prgEM.stEL3443_IO.MDP5001_341_Input.MDP5001_341_L1_Status_Voltage_Sign_Bit 		:= MDP5001_341_L1_Status_Voltage_Sign_Bit;
prgEM.stEL3443_IO.MDP5001_341_Input.MDP5001_341_L1_Status_Overvoltage			:= MDP5001_341_L1_Status_Overvoltage;
prgEM.stEL3443_IO.MDP5001_341_Input.MDP5001_341_L1_Status_Overcurrent			:= MDP5001_341_L1_Status_Overcurrent;
prgEM.stEL3443_IO.MDP5001_341_Input.MDP5001_341_L1_Status_Inaccurate_Voltage	:= MDP5001_341_L1_Status_Inaccurate_Voltage;
prgEM.stEL3443_IO.MDP5001_341_Input.MDP5001_341_L1_Status_Inaccurate_Current	:= MDP5001_341_L1_Status_Inaccurate_Current;
prgEM.stEL3443_IO.MDP5001_341_Input.MDP5001_341_L1_Status_Voltage_Guard_Warning	:= MDP5001_341_L1_Status_Voltage_Guard_Warning;
prgEM.stEL3443_IO.MDP5001_341_Input.MDP5001_341_L1_Status_Voltage_Guard_Error	:= MDP5001_341_L1_Status_Voltage_Guard_Error;
prgEM.stEL3443_IO.MDP5001_341_Input.MDP5001_341_L1_Status_Current_Guard_Warning	:= MDP5001_341_L1_Status_Current_Guard_Warning;
prgEM.stEL3443_IO.MDP5001_341_Input.MDP5001_341_L1_Status_Current_Guard_Error	:= MDP5001_341_L1_Status_Current_Guard_Error;
prgEM.stEL3443_IO.MDP5001_341_Input.MDP5001_341_L1_Status_TxPDO_Toggle			:= MDP5001_341_L1_Status_TxPDO_Toggle;
prgEM.stEL3443_IO.MDP5001_341_Input.MDP5001_341_L1_Basic_Voltage				:= MDP5001_341_L1_Basic_Voltage;
prgEM.stEL3443_IO.MDP5001_341_Input.MDP5001_341_L1_Basic_Current				:= MDP5001_341_L1_Basic_Current;
prgEM.stEL3443_IO.MDP5001_341_Input.MDP5001_341_L1_Power_Active_Power			:= MDP5001_341_L1_Power_Active_Power;
prgEM.stEL3443_IO.MDP5001_341_Input.MDP5001_341_L1_Power_Apparent_Power			:= MDP5001_341_L1_Power_Apparent_Power;
prgEM.stEL3443_IO.MDP5001_341_Input.MDP5001_341_L1_Power_Reactive_Power			:= MDP5001_341_L1_Power_Reactive_Power;
prgEM.stEL3443_IO.MDP5001_341_Input.MDP5001_341_L1_Power_Power_Factor			:= MDP5001_341_L1_Power_Power_Factor;
prgEM.stEL3443_IO.MDP5001_341_Input.MDP5001_341_L2_Status_Voltage_Sign_Bit 		:= MDP5001_341_L2_Status_Voltage_Sign_Bit;
prgEM.stEL3443_IO.MDP5001_341_Input.MDP5001_341_L2_Status_Overvoltage			:= MDP5001_341_L2_Status_Overvoltage;
prgEM.stEL3443_IO.MDP5001_341_Input.MDP5001_341_L2_Status_Overcurrent			:= MDP5001_341_L2_Status_Overcurrent;
prgEM.stEL3443_IO.MDP5001_341_Input.MDP5001_341_L2_Status_Inaccurate_Voltage	:= MDP5001_341_L2_Status_Inaccurate_Voltage;
prgEM.stEL3443_IO.MDP5001_341_Input.MDP5001_341_L2_Status_Inaccurate_Current	:= MDP5001_341_L2_Status_Inaccurate_Current;
prgEM.stEL3443_IO.MDP5001_341_Input.MDP5001_341_L2_Status_Voltage_Guard_Warning	:= MDP5001_341_L2_Status_Voltage_Guard_Warning;
prgEM.stEL3443_IO.MDP5001_341_Input.MDP5001_341_L2_Status_Voltage_Guard_Error	:= MDP5001_341_L2_Status_Voltage_Guard_Error;
prgEM.stEL3443_IO.MDP5001_341_Input.MDP5001_341_L2_Status_Current_Guard_Warning	:= MDP5001_341_L2_Status_Current_Guard_Warning;
prgEM.stEL3443_IO.MDP5001_341_Input.MDP5001_341_L2_Status_Current_Guard_Error	:= MDP5001_341_L2_Status_Current_Guard_Error;
prgEM.stEL3443_IO.MDP5001_341_Input.MDP5001_341_L2_Status_TxPDO_Toggle			:= MDP5001_341_L2_Status_TxPDO_Toggle;
prgEM.stEL3443_IO.MDP5001_341_Input.MDP5001_341_L2_Basic_Voltage				:= MDP5001_341_L2_Basic_Voltage;
prgEM.stEL3443_IO.MDP5001_341_Input.MDP5001_341_L2_Basic_Current				:= MDP5001_341_L2_Basic_Current;
prgEM.stEL3443_IO.MDP5001_341_Input.MDP5001_341_L2_Power_Active_Power			:= MDP5001_341_L2_Power_Active_Power;
prgEM.stEL3443_IO.MDP5001_341_Input.MDP5001_341_L2_Power_Apparent_Power			:= MDP5001_341_L2_Power_Apparent_Power;
prgEM.stEL3443_IO.MDP5001_341_Input.MDP5001_341_L2_Power_Reactive_Power			:= MDP5001_341_L2_Power_Reactive_Power;
prgEM.stEL3443_IO.MDP5001_341_Input.MDP5001_341_L2_Power_Power_Factor			:= MDP5001_341_L2_Power_Power_Factor;
prgEM.stEL3443_IO.MDP5001_341_Input.MDP5001_341_L3_Status_Voltage_Sign_Bit 		:= MDP5001_341_L3_Status_Voltage_Sign_Bit;
prgEM.stEL3443_IO.MDP5001_341_Input.MDP5001_341_L3_Status_Overvoltage			:= MDP5001_341_L3_Status_Overvoltage;
prgEM.stEL3443_IO.MDP5001_341_Input.MDP5001_341_L3_Status_Overcurrent			:= MDP5001_341_L3_Status_Overcurrent;
prgEM.stEL3443_IO.MDP5001_341_Input.MDP5001_341_L3_Status_Inaccurate_Voltage	:= MDP5001_341_L3_Status_Inaccurate_Voltage;
prgEM.stEL3443_IO.MDP5001_341_Input.MDP5001_341_L3_Status_Inaccurate_Current	:= MDP5001_341_L3_Status_Inaccurate_Current;
prgEM.stEL3443_IO.MDP5001_341_Input.MDP5001_341_L3_Status_Voltage_Guard_Warning	:= MDP5001_341_L3_Status_Voltage_Guard_Warning;
prgEM.stEL3443_IO.MDP5001_341_Input.MDP5001_341_L3_Status_Voltage_Guard_Error	:= MDP5001_341_L3_Status_Voltage_Guard_Error;
prgEM.stEL3443_IO.MDP5001_341_Input.MDP5001_341_L3_Status_Current_Guard_Warning	:= MDP5001_341_L3_Status_Current_Guard_Warning;
prgEM.stEL3443_IO.MDP5001_341_Input.MDP5001_341_L3_Status_Current_Guard_Error	:= MDP5001_341_L3_Status_Current_Guard_Error;
prgEM.stEL3443_IO.MDP5001_341_Input.MDP5001_341_L3_Status_TxPDO_Toggle			:= MDP5001_341_L3_Status_TxPDO_Toggle;
prgEM.stEL3443_IO.MDP5001_341_Input.MDP5001_341_L3_Basic_Voltage				:= MDP5001_341_L3_Basic_Voltage;
prgEM.stEL3443_IO.MDP5001_341_Input.MDP5001_341_L3_Basic_Current				:= MDP5001_341_L3_Basic_Current;
prgEM.stEL3443_IO.MDP5001_341_Input.MDP5001_341_L3_Power_Active_Power			:= MDP5001_341_L3_Power_Active_Power;
prgEM.stEL3443_IO.MDP5001_341_Input.MDP5001_341_L3_Power_Apparent_Power			:= MDP5001_341_L3_Power_Apparent_Power;
prgEM.stEL3443_IO.MDP5001_341_Input.MDP5001_341_L3_Power_Reactive_Power			:= MDP5001_341_L3_Power_Reactive_Power;
prgEM.stEL3443_IO.MDP5001_341_Input.MDP5001_341_L3_Power_Power_Factor			:= MDP5001_341_L3_Power_Power_Factor;
prgEM.stEL3443_IO.MDP5001_341_Input.MDP5001_341_Total_Status_System_State		:= MDP5001_341_Total_Status_System_State  ;	
prgEM.stEL3443_IO.MDP5001_341_Input.MDP5001_341_Total_Status_Grid_Direction		:= MDP5001_341_Total_Status_Grid_Direction ;
prgEM.stEL3443_IO.MDP5001_341_Input.MDP5001_341_Total_Status_Frequency_Guard_Warning 		:= MDP5001_341_Total_Status_Frequency_Guard_Warning ;
prgEM.stEL3443_IO.MDP5001_341_Input.MDP5001_341_Total_Status_Frequency_Guard_Error 			:= MDP5001_341_Total_Status_Frequency_Guard_Error  ;
prgEM.stEL3443_IO.MDP5001_341_Input.MDP5001_341_Total_Status_Neutral_Current_Guard_Warning	:= MDP5001_341_Total_Status_Neutral_Current_Guard_Warning ;
prgEM.stEL3443_IO.MDP5001_341_Input.MDP5001_341_Total_Status_Neutral_Current_Guard_Error	:= MDP5001_341_Total_Status_Neutral_Current_Guard_Error;
prgEM.stEL3443_IO.MDP5001_341_Input.MDP5001_341_Total_Status_Active_Power_Guard_Warning		:= MDP5001_341_Total_Status_Active_Power_Guard_Warning ;
prgEM.stEL3443_IO.MDP5001_341_Input.MDP5001_341_Total_Status_Active_Power_Guard_Error		:= MDP5001_341_Total_Status_Active_Power_Guard_Error ;
prgEM.stEL3443_IO.MDP5001_341_Input.MDP5001_341_Total_Status_Apparent_Power_Guard_Warning	:= MDP5001_341_Total_Status_Apparent_Power_Guard_Warning ;
prgEM.stEL3443_IO.MDP5001_341_Input.MDP5001_341_Total_Status_Apparent_Power_Guard_Error		:= MDP5001_341_Total_Status_Apparent_Power_Guard_Error ;
prgEM.stEL3443_IO.MDP5001_341_Input.MDP5001_341_Total_Status_Power_Quality_Guard_Warning	:= MDP5001_341_Total_Status_Power_Quality_Guard_Warning ;
prgEM.stEL3443_IO.MDP5001_341_Input.MDP5001_341_Total_Status_Power_Quality_Guard_Error		:= MDP5001_341_Total_Status_Power_Quality_Guard_Error ;
prgEM.stEL3443_IO.MDP5001_341_Input.MDP5001_341_Total_Status_TxPDO_State					:= MDP5001_341_Total_Status_TxPDO_State ;
prgEM.stEL3443_IO.MDP5001_341_Input.MDP5001_341_Total_Status_TxPDO_Toggle					:= MDP5001_341_Total_Status_TxPDO_Toggle ;
prgEM.stEL3443_IO.MDP5001_341_Input.MDP5001_341_Total_Status_Power_Quality_Factor			:= MDP5001_341_Total_Status_Power_Quality_Factor ;
prgEM.stEL3443_IO.MDP5001_341_Input.MDP5001_341_Total_Basic_Frequency						:= MDP5001_341_Total_Basic_Frequency;
prgEM.stEL3443_IO.MDP5001_341_Input.MDP5001_341_Total_Basic_Power_Factor					:= MDP5001_341_Total_Basic_Power_Factor  ;
prgEM.stEL3443_IO.MDP5001_341_Input.MDP5001_341_Total_Basic_Calculated_Neutral_Line_Current	:= MDP5001_341_Total_Basic_Calculated_Neutral_Line_Current ;
prgEM.stEL3443_IO.MDP5001_341_Input.MDP5001_341_Total_Variant_Value_In_TxPDO_Toggle			:= MDP5001_341_Total_Variant_Value_In_TxPDO_Toggle ;
prgEM.stEL3443_IO.MDP5001_341_Input.MDP5001_341_Total_Variant_Value_In_Index_1_REAL			:= MDP5001_341_Total_Variant_Value_In_Index_1_REAL ;
prgEM.stEL3443_IO.MDP5001_341_Input.MDP5001_341_Total_Variant_Value_In_Value_1_REAL			:= MDP5001_341_Total_Variant_Value_In_Value_1_REAL ;
prgEM.stEL3443_IO.MDP5001_341_Input.MDP5001_341_Total_Variant_Value_In_Index_2_REAL			:= MDP5001_341_Total_Variant_Value_In_Index_2_REAL ;
prgEM.stEL3443_IO.MDP5001_341_Input.MDP5001_341_Total_Variant_Value_In_Value_2_REAL			:= MDP5001_341_Total_Variant_Value_In_Value_2_REAL ;
prgEM.stEL3443_IO.MDP5001_341_Input.MDP5001_341_Total_Variant_Value_In_Index_3_REAL			:= MDP5001_341_Total_Variant_Value_In_Index_3_REAL ;
prgEM.stEL3443_IO.MDP5001_341_Input.MDP5001_341_Total_Variant_Value_In_Value_3_REAL			:= MDP5001_341_Total_Variant_Value_In_Value_3_REAL ;
prgEM.stEL3443_IO.MDP5001_341_Input.MDP5001_341_Total_Variant_Value_In_Index_4_ULINT		:= MDP5001_341_Total_Variant_Value_In_Index_4_ULINT ;
prgEM.stEL3443_IO.MDP5001_341_Input.MDP5001_341_Total_Variant_Value_In_Value_4_ULINT		:= MDP5001_341_Total_Variant_Value_In_Value_4_ULINT ;
prgEM.stEL3443_IO.MDP5001_341_Input.MDP5001_341_DPM_Data_Data_1			:= MDP5001_341_DPM_Data_Data_1;
prgEM.stEL3443_IO.MDP5001_341_Input.MDP5001_341_DPM_Data_Data_2			:= MDP5001_341_DPM_Data_Data_2;
prgEM.stEL3443_IO.MDP5001_341_Input.MDP5001_341_DPM_Data_Data_3			:= MDP5001_341_DPM_Data_Data_3;
prgEM.stEL3443_IO.MDP5001_341_Input.MDP5001_341_DPM_Data_Data_4			:= MDP5001_341_DPM_Data_Data_4;
prgEM.stEL3443_IO.MDP5001_341_Input.MDP5001_341_DPM_Data_Data_5			:= MDP5001_341_DPM_Data_Data_5;
prgEM.stEL3443_IO.MDP5001_341_Input.MDP5001_341_DPM_Data_Data_6			:= MDP5001_341_DPM_Data_Data_6;
prgEM.stEL3443_IO.MDP5001_341_Input.MDP5001_341_DPM_Data_Data_7			:= MDP5001_341_DPM_Data_Data_7;
prgEM.stEL3443_IO.MDP5001_341_Input.MDP5001_341_DPM_Data_Data_8			:= MDP5001_341_DPM_Data_Data_8;
prgEM.stEL3443_IO.MDP5001_341_Input.MDP5001_341_DPM_Data_Data_9			:= MDP5001_341_DPM_Data_Data_9;
prgEM.stEL3443_IO.MDP5001_341_Input.MDP5001_341_DPM_Data_Data_10		:= MDP5001_341_DPM_Data_Data_10;
prgEM.stEL3443_IO.MDP5001_341_Input.MDP5001_341_DPM_Data_Data_11		:= MDP5001_341_DPM_Data_Data_11;
prgEM.stEL3443_IO.MDP5001_341_Input.MDP5001_341_DPM_Data_Data_12		:= MDP5001_341_DPM_Data_Data_12;
prgEM.stEL3443_IO.MDP5001_341_Input.MDP5001_341_DPM_Data_Data_13		:= MDP5001_341_DPM_Data_Data_13;
prgEM.stEL3443_IO.MDP5001_341_Input.MDP5001_341_DPM_Data_Data_14		:= MDP5001_341_DPM_Data_Data_14;
prgEM.stEL3443_IO.MDP5001_341_Input.MDP5001_341_DPM_Data_Data_15		:= MDP5001_341_DPM_Data_Data_15;
prgEM.stEL3443_IO.MDP5001_341_Input.MDP5001_341_DPM_Data_Data_16		:= MDP5001_341_DPM_Data_Data_16;
prgEM.stEL3443_IO.MDP5001_341_Input.MDP5001_341_DPM_Data_Data_17		:= MDP5001_341_DPM_Data_Data_17;
prgEM.stEL3443_IO.MDP5001_341_Input.MDP5001_341_DPM_Data_Data_18		:= MDP5001_341_DPM_Data_Data_18;
prgEM.stEL3443_IO.MDP5001_341_Input.MDP5001_341_DPM_Data_Data_19		:= MDP5001_341_DPM_Data_Data_19;
prgEM.stEL3443_IO.MDP5001_341_Input.MDP5001_341_DPM_Data_Data_20		:= MDP5001_341_DPM_Data_Data_20;
MDP5001_341_Total_Variant_Value_Out_Index_1_REAL	:= prgEM.stEL3443_IO.MDP5001_341_Output.MDP5001_341_Total_Variant_Value_Out_Index_1_REAL;
MDP5001_341_Total_Variant_Value_Out_Index_2_REAL	:= prgEM.stEL3443_IO.MDP5001_341_Output.MDP5001_341_Total_Variant_Value_Out_Index_2_REAL;
MDP5001_341_Total_Variant_Value_Out_Index_3_REAL	:= prgEM.stEL3443_IO.MDP5001_341_Output.MDP5001_341_Total_Variant_Value_Out_Index_3_REAL;
MDP5001_341_Total_Variant_Value_Out_Index_4_ULINT	:= prgEM.stEL3443_IO.MDP5001_341_Output.MDP5001_341_Total_Variant_Value_Out_Index_4_ULINT;
MDP5001_341_Total_Interval_Reset_Interval			:= prgEM.stEL3443_IO.MDP5001_341_Output.MDP5001_341_Total_Interval_Reset_Interval;

// EL3446

prgEM.stEL3446_IO.MDP5001_342_Input.MDP5001_342_I1_Channel_Overcurrent					:=	MDP5001_342_I1_Channel_Overcurrent;
prgEM.stEL3446_IO.MDP5001_342_Input.MDP5001_342_I1_Channel_Inaccurate_Current			:=	MDP5001_342_I1_Channel_Inaccurate_Current;
prgEM.stEL3446_IO.MDP5001_342_Input.MDP5001_342_I1_Channel_Current_Guard_Warning		:=	MDP5001_342_I1_Channel_Current_Guard_Warning;
prgEM.stEL3446_IO.MDP5001_342_Input.MDP5001_342_I1_Channel_Current_Guard_Error			:=	MDP5001_342_I1_Channel_Current_Guard_Error;
prgEM.stEL3446_IO.MDP5001_342_Input.MDP5001_342_I1_Channel_Apparent_Power_Guard_Warning	:=	MDP5001_342_I1_Channel_Apparent_Power_Guard_Warning;
prgEM.stEL3446_IO.MDP5001_342_Input.MDP5001_342_I1_Channel_Apparent_Power_Guard_Error	:=	MDP5001_342_I1_Channel_Apparent_Power_Guard_Error;
prgEM.stEL3446_IO.MDP5001_342_Input.MDP5001_342_I1_Channel_Active_Power_Guard_Warning	:=	MDP5001_342_I1_Channel_Active_Power_Guard_Warning;
prgEM.stEL3446_IO.MDP5001_342_Input.MDP5001_342_I1_Channel_Active_Power_Guard_Error		:=	MDP5001_342_I1_Channel_Active_Power_Guard_Error;
prgEM.stEL3446_IO.MDP5001_342_Input.MDP5001_342_I1_Channel_Reactive_Power_Guard_Warning	:=	MDP5001_342_I1_Channel_Reactive_Power_Guard_Warning;
prgEM.stEL3446_IO.MDP5001_342_Input.MDP5001_342_I1_Channel_Reactive_Power_Guard_Error	:=	MDP5001_342_I1_Channel_Reactive_Power_Guard_Error;
prgEM.stEL3446_IO.MDP5001_342_Input.MDP5001_342_I1_Channel_DPM_Inaccurate				:=	MDP5001_342_I1_Channel_DPM_Inaccurate;
prgEM.stEL3446_IO.MDP5001_342_Input.MDP5001_342_I1_Channel_DPM_Timeout					:=	MDP5001_342_I1_Channel_DPM_Timeout;
prgEM.stEL3446_IO.MDP5001_342_Input.MDP5001_342_I1_Channel_TxPDO_Toggle					:=	MDP5001_342_I1_Channel_TxPDO_Toggle;
prgEM.stEL3446_IO.MDP5001_342_Input.MDP5001_342_I1_Channel_Current						:=	MDP5001_342_I1_Channel_Current;
prgEM.stEL3446_IO.MDP5001_342_Input.MDP5001_342_I1_Channel_Active_Power					:=	MDP5001_342_I1_Channel_Active_Power;
prgEM.stEL3446_IO.MDP5001_342_Input.MDP5001_342_I1_Channel_Apparent_Power				:=	MDP5001_342_I1_Channel_Apparent_Power;
prgEM.stEL3446_IO.MDP5001_342_Input.MDP5001_342_I1_Channel_Reactive_Power_Fundamental	:=	MDP5001_342_I1_Channel_Reactive_Power_Fundamental;
prgEM.stEL3446_IO.MDP5001_342_Input.MDP5001_342_I1_Channel_Active_Energy				:=	MDP5001_342_I1_Channel_Active_Energy;
prgEM.stEL3446_IO.MDP5001_342_Input.MDP5001_342_I2_Channel_Overcurrent					:=	MDP5001_342_I2_Channel_Overcurrent;
prgEM.stEL3446_IO.MDP5001_342_Input.MDP5001_342_I2_Channel_Inaccurate_Current			:=	MDP5001_342_I2_Channel_Inaccurate_Current;
prgEM.stEL3446_IO.MDP5001_342_Input.MDP5001_342_I2_Channel_Current_Guard_Warning		:=	MDP5001_342_I2_Channel_Current_Guard_Warning;
prgEM.stEL3446_IO.MDP5001_342_Input.MDP5001_342_I2_Channel_Current_Guard_Error			:=	MDP5001_342_I2_Channel_Current_Guard_Error;
prgEM.stEL3446_IO.MDP5001_342_Input.MDP5001_342_I2_Channel_Apparent_Power_Guard_Warning	:=	MDP5001_342_I2_Channel_Apparent_Power_Guard_Warning;
prgEM.stEL3446_IO.MDP5001_342_Input.MDP5001_342_I2_Channel_Apparent_Power_Guard_Error	:=	MDP5001_342_I2_Channel_Apparent_Power_Guard_Error;
prgEM.stEL3446_IO.MDP5001_342_Input.MDP5001_342_I2_Channel_Active_Power_Guard_Warning	:=	MDP5001_342_I2_Channel_Active_Power_Guard_Warning;
prgEM.stEL3446_IO.MDP5001_342_Input.MDP5001_342_I2_Channel_Active_Power_Guard_Error		:=	MDP5001_342_I2_Channel_Active_Power_Guard_Error;
prgEM.stEL3446_IO.MDP5001_342_Input.MDP5001_342_I2_Channel_Reactive_Power_Guard_Warning	:=	MDP5001_342_I2_Channel_Reactive_Power_Guard_Warning;
prgEM.stEL3446_IO.MDP5001_342_Input.MDP5001_342_I2_Channel_Reactive_Power_Guard_Error	:=	MDP5001_342_I2_Channel_Reactive_Power_Guard_Error;
prgEM.stEL3446_IO.MDP5001_342_Input.MDP5001_342_I2_Channel_DPM_Inaccurate				:=	MDP5001_342_I2_Channel_DPM_Inaccurate;
prgEM.stEL3446_IO.MDP5001_342_Input.MDP5001_342_I2_Channel_DPM_Timeout					:=	MDP5001_342_I2_Channel_DPM_Timeout;
prgEM.stEL3446_IO.MDP5001_342_Input.MDP5001_342_I2_Channel_TxPDO_Toggle					:=	MDP5001_342_I2_Channel_TxPDO_Toggle;
prgEM.stEL3446_IO.MDP5001_342_Input.MDP5001_342_I2_Channel_Current						:=	MDP5001_342_I2_Channel_Current;
prgEM.stEL3446_IO.MDP5001_342_Input.MDP5001_342_I2_Channel_Active_Power					:=	MDP5001_342_I2_Channel_Active_Power;
prgEM.stEL3446_IO.MDP5001_342_Input.MDP5001_342_I2_Channel_Apparent_Power				:=	MDP5001_342_I2_Channel_Apparent_Power;
prgEM.stEL3446_IO.MDP5001_342_Input.MDP5001_342_I2_Channel_Reactive_Power_Fundamental	:=	MDP5001_342_I2_Channel_Reactive_Power_Fundamental;
prgEM.stEL3446_IO.MDP5001_342_Input.MDP5001_342_I2_Channel_Active_Energy				:=	MDP5001_342_I2_Channel_Active_Energy;
prgEM.stEL3446_IO.MDP5001_342_Input.MDP5001_342_I3_Channel_Overcurrent					:=	MDP5001_342_I3_Channel_Overcurrent;
prgEM.stEL3446_IO.MDP5001_342_Input.MDP5001_342_I3_Channel_Inaccurate_Current			:=	MDP5001_342_I3_Channel_Inaccurate_Current;
prgEM.stEL3446_IO.MDP5001_342_Input.MDP5001_342_I3_Channel_Current_Guard_Warning		:=	MDP5001_342_I3_Channel_Current_Guard_Warning;
prgEM.stEL3446_IO.MDP5001_342_Input.MDP5001_342_I3_Channel_Current_Guard_Error			:=	MDP5001_342_I3_Channel_Current_Guard_Error;
prgEM.stEL3446_IO.MDP5001_342_Input.MDP5001_342_I3_Channel_Apparent_Power_Guard_Warning	:=	MDP5001_342_I3_Channel_Apparent_Power_Guard_Warning;
prgEM.stEL3446_IO.MDP5001_342_Input.MDP5001_342_I3_Channel_Apparent_Power_Guard_Error	:=	MDP5001_342_I3_Channel_Apparent_Power_Guard_Error;
prgEM.stEL3446_IO.MDP5001_342_Input.MDP5001_342_I3_Channel_Active_Power_Guard_Warning	:=	MDP5001_342_I3_Channel_Active_Power_Guard_Warning;
prgEM.stEL3446_IO.MDP5001_342_Input.MDP5001_342_I3_Channel_Active_Power_Guard_Error		:=	MDP5001_342_I3_Channel_Active_Power_Guard_Error;
prgEM.stEL3446_IO.MDP5001_342_Input.MDP5001_342_I3_Channel_Reactive_Power_Guard_Warning	:=	MDP5001_342_I3_Channel_Reactive_Power_Guard_Warning;
prgEM.stEL3446_IO.MDP5001_342_Input.MDP5001_342_I3_Channel_Reactive_Power_Guard_Error	:=	MDP5001_342_I3_Channel_Reactive_Power_Guard_Error;
prgEM.stEL3446_IO.MDP5001_342_Input.MDP5001_342_I3_Channel_DPM_Inaccurate				:=	MDP5001_342_I3_Channel_DPM_Inaccurate;
prgEM.stEL3446_IO.MDP5001_342_Input.MDP5001_342_I3_Channel_DPM_Timeout					:=	MDP5001_342_I3_Channel_DPM_Timeout;
prgEM.stEL3446_IO.MDP5001_342_Input.MDP5001_342_I3_Channel_TxPDO_Toggle					:=	MDP5001_342_I3_Channel_TxPDO_Toggle;
prgEM.stEL3446_IO.MDP5001_342_Input.MDP5001_342_I3_Channel_Current						:=	MDP5001_342_I3_Channel_Current;
prgEM.stEL3446_IO.MDP5001_342_Input.MDP5001_342_I3_Channel_Active_Power					:=	MDP5001_342_I3_Channel_Active_Power;
prgEM.stEL3446_IO.MDP5001_342_Input.MDP5001_342_I3_Channel_Apparent_Power				:=	MDP5001_342_I3_Channel_Apparent_Power;
prgEM.stEL3446_IO.MDP5001_342_Input.MDP5001_342_I3_Channel_Reactive_Power_Fundamental	:=	MDP5001_342_I3_Channel_Reactive_Power_Fundamental;
prgEM.stEL3446_IO.MDP5001_342_Input.MDP5001_342_I3_Channel_Active_Energy				:=	MDP5001_342_I3_Channel_Active_Energy;
prgEM.stEL3446_IO.MDP5001_342_Input.MDP5001_342_I4_Channel_Overcurrent					:=	MDP5001_342_I4_Channel_Overcurrent;
prgEM.stEL3446_IO.MDP5001_342_Input.MDP5001_342_I4_Channel_Inaccurate_Current			:=	MDP5001_342_I4_Channel_Inaccurate_Current;
prgEM.stEL3446_IO.MDP5001_342_Input.MDP5001_342_I4_Channel_Current_Guard_Warning		:=	MDP5001_342_I4_Channel_Current_Guard_Warning;
prgEM.stEL3446_IO.MDP5001_342_Input.MDP5001_342_I4_Channel_Current_Guard_Error			:=	MDP5001_342_I4_Channel_Current_Guard_Error;
prgEM.stEL3446_IO.MDP5001_342_Input.MDP5001_342_I4_Channel_Apparent_Power_Guard_Warning	:=	MDP5001_342_I4_Channel_Apparent_Power_Guard_Warning;
prgEM.stEL3446_IO.MDP5001_342_Input.MDP5001_342_I4_Channel_Apparent_Power_Guard_Error	:=	MDP5001_342_I4_Channel_Apparent_Power_Guard_Error;
prgEM.stEL3446_IO.MDP5001_342_Input.MDP5001_342_I4_Channel_Active_Power_Guard_Warning	:=	MDP5001_342_I4_Channel_Active_Power_Guard_Warning;
prgEM.stEL3446_IO.MDP5001_342_Input.MDP5001_342_I4_Channel_Active_Power_Guard_Error		:=	MDP5001_342_I4_Channel_Active_Power_Guard_Error;
prgEM.stEL3446_IO.MDP5001_342_Input.MDP5001_342_I4_Channel_Reactive_Power_Guard_Warning	:=	MDP5001_342_I4_Channel_Reactive_Power_Guard_Warning;
prgEM.stEL3446_IO.MDP5001_342_Input.MDP5001_342_I4_Channel_Reactive_Power_Guard_Error	:=	MDP5001_342_I4_Channel_Reactive_Power_Guard_Error;
prgEM.stEL3446_IO.MDP5001_342_Input.MDP5001_342_I4_Channel_DPM_Inaccurate				:=	MDP5001_342_I4_Channel_DPM_Inaccurate;
prgEM.stEL3446_IO.MDP5001_342_Input.MDP5001_342_I4_Channel_DPM_Timeout					:=	MDP5001_342_I4_Channel_DPM_Timeout;
prgEM.stEL3446_IO.MDP5001_342_Input.MDP5001_342_I4_Channel_TxPDO_Toggle					:=	MDP5001_342_I4_Channel_TxPDO_Toggle;
prgEM.stEL3446_IO.MDP5001_342_Input.MDP5001_342_I4_Channel_Current						:=	MDP5001_342_I4_Channel_Current;
prgEM.stEL3446_IO.MDP5001_342_Input.MDP5001_342_I4_Channel_Active_Power					:=	MDP5001_342_I4_Channel_Active_Power;
prgEM.stEL3446_IO.MDP5001_342_Input.MDP5001_342_I4_Channel_Apparent_Power				:=	MDP5001_342_I4_Channel_Apparent_Power;
prgEM.stEL3446_IO.MDP5001_342_Input.MDP5001_342_I4_Channel_Reactive_Power_Fundamental	:=	MDP5001_342_I4_Channel_Reactive_Power_Fundamental;
prgEM.stEL3446_IO.MDP5001_342_Input.MDP5001_342_I4_Channel_Active_Energy				:=	MDP5001_342_I4_Channel_Active_Energy;
prgEM.stEL3446_IO.MDP5001_342_Input.MDP5001_342_I5_Channel_Overcurrent					:=	MDP5001_342_I5_Channel_Overcurrent;
prgEM.stEL3446_IO.MDP5001_342_Input.MDP5001_342_I5_Channel_Inaccurate_Current			:=	MDP5001_342_I5_Channel_Inaccurate_Current;
prgEM.stEL3446_IO.MDP5001_342_Input.MDP5001_342_I5_Channel_Current_Guard_Warning		:=	MDP5001_342_I5_Channel_Current_Guard_Warning;
prgEM.stEL3446_IO.MDP5001_342_Input.MDP5001_342_I5_Channel_Current_Guard_Error			:=	MDP5001_342_I5_Channel_Current_Guard_Error;
prgEM.stEL3446_IO.MDP5001_342_Input.MDP5001_342_I5_Channel_Apparent_Power_Guard_Warning	:=	MDP5001_342_I5_Channel_Apparent_Power_Guard_Warning;
prgEM.stEL3446_IO.MDP5001_342_Input.MDP5001_342_I5_Channel_Apparent_Power_Guard_Error	:=	MDP5001_342_I5_Channel_Apparent_Power_Guard_Error;
prgEM.stEL3446_IO.MDP5001_342_Input.MDP5001_342_I5_Channel_Active_Power_Guard_Warning	:=	MDP5001_342_I5_Channel_Active_Power_Guard_Warning;
prgEM.stEL3446_IO.MDP5001_342_Input.MDP5001_342_I5_Channel_Active_Power_Guard_Error		:=	MDP5001_342_I5_Channel_Active_Power_Guard_Error;
prgEM.stEL3446_IO.MDP5001_342_Input.MDP5001_342_I5_Channel_Reactive_Power_Guard_Warning	:=	MDP5001_342_I5_Channel_Reactive_Power_Guard_Warning;
prgEM.stEL3446_IO.MDP5001_342_Input.MDP5001_342_I5_Channel_Reactive_Power_Guard_Error	:=	MDP5001_342_I5_Channel_Reactive_Power_Guard_Error;
prgEM.stEL3446_IO.MDP5001_342_Input.MDP5001_342_I5_Channel_DPM_Inaccurate				:=	MDP5001_342_I5_Channel_DPM_Inaccurate;
prgEM.stEL3446_IO.MDP5001_342_Input.MDP5001_342_I5_Channel_DPM_Timeout					:=	MDP5001_342_I5_Channel_DPM_Timeout;
prgEM.stEL3446_IO.MDP5001_342_Input.MDP5001_342_I5_Channel_TxPDO_Toggle					:=	MDP5001_342_I5_Channel_TxPDO_Toggle;
prgEM.stEL3446_IO.MDP5001_342_Input.MDP5001_342_I5_Channel_Current						:=	MDP5001_342_I5_Channel_Current;
prgEM.stEL3446_IO.MDP5001_342_Input.MDP5001_342_I5_Channel_Active_Power					:=	MDP5001_342_I5_Channel_Active_Power;
prgEM.stEL3446_IO.MDP5001_342_Input.MDP5001_342_I5_Channel_Apparent_Power				:=	MDP5001_342_I5_Channel_Apparent_Power;
prgEM.stEL3446_IO.MDP5001_342_Input.MDP5001_342_I5_Channel_Reactive_Power_Fundamental	:=	MDP5001_342_I5_Channel_Reactive_Power_Fundamental;
prgEM.stEL3446_IO.MDP5001_342_Input.MDP5001_342_I5_Channel_Active_Energy				:=	MDP5001_342_I5_Channel_Active_Energy;
prgEM.stEL3446_IO.MDP5001_342_Input.MDP5001_342_I6_Channel_Overcurrent					:=	MDP5001_342_I6_Channel_Overcurrent;
prgEM.stEL3446_IO.MDP5001_342_Input.MDP5001_342_I6_Channel_Inaccurate_Current			:=	MDP5001_342_I6_Channel_Inaccurate_Current;
prgEM.stEL3446_IO.MDP5001_342_Input.MDP5001_342_I6_Channel_Current_Guard_Warning		:=	MDP5001_342_I6_Channel_Current_Guard_Warning;
prgEM.stEL3446_IO.MDP5001_342_Input.MDP5001_342_I6_Channel_Current_Guard_Error			:=	MDP5001_342_I6_Channel_Current_Guard_Error;
prgEM.stEL3446_IO.MDP5001_342_Input.MDP5001_342_I6_Channel_Apparent_Power_Guard_Warning	:=	MDP5001_342_I6_Channel_Apparent_Power_Guard_Warning;
prgEM.stEL3446_IO.MDP5001_342_Input.MDP5001_342_I6_Channel_Apparent_Power_Guard_Error	:=	MDP5001_342_I6_Channel_Apparent_Power_Guard_Error;
prgEM.stEL3446_IO.MDP5001_342_Input.MDP5001_342_I6_Channel_Active_Power_Guard_Warning	:=	MDP5001_342_I6_Channel_Active_Power_Guard_Warning;
prgEM.stEL3446_IO.MDP5001_342_Input.MDP5001_342_I6_Channel_Active_Power_Guard_Error		:=	MDP5001_342_I6_Channel_Active_Power_Guard_Error;
prgEM.stEL3446_IO.MDP5001_342_Input.MDP5001_342_I6_Channel_Reactive_Power_Guard_Warning	:=	MDP5001_342_I6_Channel_Reactive_Power_Guard_Warning;
prgEM.stEL3446_IO.MDP5001_342_Input.MDP5001_342_I6_Channel_Reactive_Power_Guard_Error	:=	MDP5001_342_I6_Channel_Reactive_Power_Guard_Error;
prgEM.stEL3446_IO.MDP5001_342_Input.MDP5001_342_I6_Channel_DPM_Inaccurate				:=	MDP5001_342_I6_Channel_DPM_Inaccurate;
prgEM.stEL3446_IO.MDP5001_342_Input.MDP5001_342_I6_Channel_DPM_Timeout					:=	MDP5001_342_I6_Channel_DPM_Timeout;
prgEM.stEL3446_IO.MDP5001_342_Input.MDP5001_342_I6_Channel_TxPDO_Toggle					:=	MDP5001_342_I6_Channel_TxPDO_Toggle;
prgEM.stEL3446_IO.MDP5001_342_Input.MDP5001_342_I6_Channel_Current						:=	MDP5001_342_I6_Channel_Current;
prgEM.stEL3446_IO.MDP5001_342_Input.MDP5001_342_I6_Channel_Active_Power					:=	MDP5001_342_I6_Channel_Active_Power;
prgEM.stEL3446_IO.MDP5001_342_Input.MDP5001_342_I6_Channel_Apparent_Power				:=	MDP5001_342_I6_Channel_Apparent_Power;
prgEM.stEL3446_IO.MDP5001_342_Input.MDP5001_342_I6_Channel_Reactive_Power_Fundamental	:=	MDP5001_342_I6_Channel_Reactive_Power_Fundamental;
prgEM.stEL3446_IO.MDP5001_342_Input.MDP5001_342_I6_Channel_Active_Energy				:=	MDP5001_342_I6_Channel_Active_Energy;
prgEM.stEL3446_IO.MDP5001_342_Input.MDP5001_342_DPM_Variant_Value_In_TxPDO_Toggle		:=	MDP5001_342_DPM_Variant_Value_In_TxPDO_Toggle;
prgEM.stEL3446_IO.MDP5001_342_Input.MDP5001_342_DPM_Variant_Value_In_Index_1_REAL		:=	MDP5001_342_DPM_Variant_Value_In_Index_1_REAL;
prgEM.stEL3446_IO.MDP5001_342_Input.MDP5001_342_DPM_Variant_Value_In_Value_1_REAL		:=	MDP5001_342_DPM_Variant_Value_In_Value_1_REAL;
prgEM.stEL3446_IO.MDP5001_342_Input.MDP5001_342_DPM_Variant_Value_In_Index_2_REAL		:=	MDP5001_342_DPM_Variant_Value_In_Index_2_REAL;
prgEM.stEL3446_IO.MDP5001_342_Input.MDP5001_342_DPM_Variant_Value_In_Value_2_REAL		:=	MDP5001_342_DPM_Variant_Value_In_Value_2_REAL;
prgEM.stEL3446_IO.MDP5001_342_Input.MDP5001_342_DPM_Variant_Value_In_Index_3_REAL		:=	MDP5001_342_DPM_Variant_Value_In_Index_3_REAL;
prgEM.stEL3446_IO.MDP5001_342_Input.MDP5001_342_DPM_Variant_Value_In_Value_3_REAL		:=	MDP5001_342_DPM_Variant_Value_In_Value_3_REAL;
prgEM.stEL3446_IO.MDP5001_342_Input.MDP5001_342_DPM_Variant_Value_In_Index_4_ULINT		:=	MDP5001_342_DPM_Variant_Value_In_Index_4_ULINT;
prgEM.stEL3446_IO.MDP5001_342_Input.MDP5001_342_DPM_Variant_Value_In_Value_4_ULINT		:=	MDP5001_342_DPM_Variant_Value_In_Value_4_ULINT;
MDP5001_342_DPM_Variant_Value_Out_Index_1_REAL	:= 		prgEM.stEL3446_IO.MDP5001_342_Output.MDP5001_342_DPM_Variant_Value_Out_Index_1_REAL	;
MDP5001_342_DPM_Variant_Value_Out_Index_2_REAL	:= 		prgEM.stEL3446_IO.MDP5001_342_Output.MDP5001_342_DPM_Variant_Value_Out_Index_2_REAL	;	
MDP5001_342_DPM_Variant_Value_Out_Index_3_REAL	:= 		prgEM.stEL3446_IO.MDP5001_342_Output.MDP5001_342_DPM_Variant_Value_Out_Index_3_REAL	;
MDP5001_342_DPM_Variant_Value_Out_Index_4_ULINT	:= 		prgEM.stEL3446_IO.MDP5001_342_Output.MDP5001_342_DPM_Variant_Value_Out_Index_4_ULINT	;
MDP5001_342_DPM_Data_Data_1						:= 		prgEM.stEL3446_IO.MDP5001_342_Output.MDP5001_342_DPM_Data_Data_1	;
MDP5001_342_DPM_Data_Data_2						:= 		prgEM.stEL3446_IO.MDP5001_342_Output.MDP5001_342_DPM_Data_Data_2	;
MDP5001_342_DPM_Data_Data_3						:= 		prgEM.stEL3446_IO.MDP5001_342_Output.MDP5001_342_DPM_Data_Data_3	;
MDP5001_342_DPM_Data_Data_4						:= 		prgEM.stEL3446_IO.MDP5001_342_Output.MDP5001_342_DPM_Data_Data_4	;
MDP5001_342_DPM_Data_Data_5						:= 		prgEM.stEL3446_IO.MDP5001_342_Output.MDP5001_342_DPM_Data_Data_5	;
MDP5001_342_DPM_Data_Data_6						:= 		prgEM.stEL3446_IO.MDP5001_342_Output.MDP5001_342_DPM_Data_Data_6	;
MDP5001_342_DPM_Data_Data_7						:= 		prgEM.stEL3446_IO.MDP5001_342_Output.MDP5001_342_DPM_Data_Data_7	;
MDP5001_342_DPM_Data_Data_8						:= 		prgEM.stEL3446_IO.MDP5001_342_Output.MDP5001_342_DPM_Data_Data_8	;
MDP5001_342_DPM_Data_Data_9						:= 		prgEM.stEL3446_IO.MDP5001_342_Output.MDP5001_342_DPM_Data_Data_9	;
MDP5001_342_DPM_Data_Data_10					:= 		prgEM.stEL3446_IO.MDP5001_342_Output.MDP5001_342_DPM_Data_Data_10	;
MDP5001_342_DPM_Data_Data_11					:= 		prgEM.stEL3446_IO.MDP5001_342_Output.MDP5001_342_DPM_Data_Data_11	;
MDP5001_342_DPM_Data_Data_12					:= 		prgEM.stEL3446_IO.MDP5001_342_Output.MDP5001_342_DPM_Data_Data_12	;
MDP5001_342_DPM_Data_Data_13					:= 		prgEM.stEL3446_IO.MDP5001_342_Output.MDP5001_342_DPM_Data_Data_13	;
MDP5001_342_DPM_Data_Data_14					:= 		prgEM.stEL3446_IO.MDP5001_342_Output.MDP5001_342_DPM_Data_Data_14	;
MDP5001_342_DPM_Data_Data_15					:= 		prgEM.stEL3446_IO.MDP5001_342_Output.MDP5001_342_DPM_Data_Data_15	;
MDP5001_342_DPM_Data_Data_16					:= 		prgEM.stEL3446_IO.MDP5001_342_Output.MDP5001_342_DPM_Data_Data_16	;
MDP5001_342_DPM_Data_Data_17					:= 		prgEM.stEL3446_IO.MDP5001_342_Output.MDP5001_342_DPM_Data_Data_17	;
MDP5001_342_DPM_Data_Data_18					:= 		prgEM.stEL3446_IO.MDP5001_342_Output.MDP5001_342_DPM_Data_Data_18	;
MDP5001_342_DPM_Data_Data_19					:= 		prgEM.stEL3446_IO.MDP5001_342_Output.MDP5001_342_DPM_Data_Data_19	;
MDP5001_342_DPM_Data_Data_20					:= 		prgEM.stEL3446_IO.MDP5001_342_Output.MDP5001_342_DPM_Data_Data_20	;

// EL2008
b_VarOut1	:= prgEMS.b_Out_CH1;
b_VarOut2	:= prgEMS.b_Out_CH2;
b_VarOut3	:= prgEMS.b_Out_CH3;
b_VarOut4	:= prgEMS.b_Out_CH4;
b_VarOut5	:= prgEMS.b_Out_CH5;
b_VarOut6	:= prgEMS.b_Out_CH6;
b_VarOut7	:= prgEMS.b_Out_CH7;
b_VarOut8	:= prgEMS.b_Out_CH8;

//EL1008
prgEMS.b_Input_KeySwitch 	:=  b_VarIn1;
prgEMS.b_Input_Spare		:= 	b_VarIn2;

END_PROGRAM

// ---- POUs/prgEM.TcPOU
PROGRAM prgEM
VAR

 	fbEL3443DPM 		: FB_EM_Beckhoff_EL3443;	//EL3443 | PDO Assignment "DPM" (DPM: Distributed Power Measurement) |3-phase power measurement terminal with extended functionality
	fb_EL3446			: FB_EM_Beckhoff_EL3446;
	lr_RealPower_Grid	: LREAL;						//{#lynus.ag#()}
	lr_ApparentPower_Grid: LREAL;						//{#lynus.ag#()}
	lr_ReactivePower_Grid: LREAL;						//{#lynus.ag#()}
	lr_Frequency_Grid	: LREAL;						//{#lynus.ag#()}

	lr_Voltage_L1N		: LREAL;						//{#lynus.ag#()}
	lr_Voltage_L2N		: LREAL;						//{#lynus.ag#()}
	lr_Voltage_L3N		: LREAL;						//{#lynus.ag#()}
	lr_Voltage_L1L2		: LREAL;						//{#lynus.ag#()}
	lr_Voltage_L2L3		: LREAL;						//{#lynus.ag#()}
	lr_Voltage_L3L1		: LREAL;						//{#lynus.ag#()}
 	lr_Current_L1		: LREAL;						//{#lynus.ag#()}
	lr_Current_L2		: LREAL;						//{#lynus.ag#()}
	lr_Current_L3		: LREAL;						//{#lynus.ag#()}

	lrPower_EM1		: LREAL;						//{#lynus.ag#()}
	lrPower_EM2		: LREAL;						//{#lynus.ag#()}
	lrPower_EM3		: LREAL;						//{#lynus.ag#()}
	lrPower_EM4		: LREAL;						//{#lynus.ag#()}
	lrPower_EM5		: LREAL;						//{#lynus.ag#()}
	lrPower_EM6		: LREAL;						//{#lynus.ag#()}
	lrPower_House	: LREAL;						//{#lynus.ag#()}
	fbCounter_House	: FB_EnergyCounter;

	m_negativePower: BOOL;							//{#lynus.ag#()}
	lrTemp_EM1		: LREAL;
	lrTemp_EM2		: LREAL;
	lrTemp_EM3		: LREAL;
	lrTemp_EM4		: LREAL;
	lrTemp_EM5		: LREAL;

	lrPowerTotal_raw_W_EM1				: LREAL;					//{#lynus.ag#()}
	lrApparentPowerTotal_raw_VA_EM1		: LREAL;					//{#lynus.ag#()}
	lrReactivePowerTotal_raw_VAr_EM1	: LREAL;					//{#lynus.ag#()}
	lrPowerTotal_raw_W_EM2				: LREAL;					//{#lynus.ag#()}
	lrApparentPowerTotal_raw_VA_EM2		: LREAL;					//{#lynus.ag#()}
	lrReactivePowerTotal_raw_VAr_EM2	: LREAL;					//{#lynus.ag#()}
	lrPowerTotal_raw_W_EM3				: LREAL;					//{#lynus.ag#()}
	lrApparentPowerTotal_raw_VA_EM3		: LREAL;					//{#lynus.ag#()}
	lrReactivePowerTotal_raw_VAr_EM3	: LREAL;					//{#lynus.ag#()}
	lrPowerTotal_raw_W_EM4				: LREAL;					//{#lynus.ag#()}
	lrApparentPowerTotal_raw_VA_EM4		: LREAL;					//{#lynus.ag#()}
	lrReactivePowerTotal_raw_VAr_EM4	: LREAL;					//{#lynus.ag#()}
	lrPowerTotal_raw_W_EM5				: LREAL;					//{#lynus.ag#()}
	lrApparentPowerTotal_raw_VA_EM5		: LREAL;					//{#lynus.ag#()}
	lrReactivePowerTotal_raw_VAr_EM5	: LREAL;					//{#lynus.ag#()}
		

END_VAR
VAR_INPUT
	ui_PhaseSelector_CH1: UINT;						//{#lynus.ag#()}
	ui_PhaseSelector_CH2: UINT;						//{#lynus.ag#()}
	ui_PhaseSelector_CH3: UINT;						//{#lynus.ag#()}
	ui_PhaseSelector_CH4: UINT;						//{#lynus.ag#()}
	ui_PhaseSelector_CH5: UINT;						//{#lynus.ag#()}
	ui_PhaseSelector_CH6: UINT:=1;						//{#lynus.ag#()}
	stEL3443_IO 						: MDP5001_341_7CD731EE;
	stEL3446_IO 						: MDP5001_342_066CA8C6; 
	b_Invers_FB3446_CH1	:BOOL;
	b_Invers_FB3446_CH2	:BOOL;
	b_Invers_FB3446_CH3	:BOOL;
	b_Invers_FB3446_CH4	:BOOL;
	b_Invers_FB3446_CH5	:BOOL;
	b_Invers_FB3446_CH6	:BOOL;
END_VAR
VAR PERSISTENT
	uiCurrentTransformerRatio	:UINT:=400;
	lr_EnergyCounter_Grid	: LREAL;						//{#lynus.ag#()}
	lr_EnergyCounter_EM1	: LREAL;						//{#lynus.ag#()}
	lr_EnergyCounter_EM2	: LREAL;						//{#lynus.ag#()}
	lr_EnergyCounter_EM3	: LREAL;						//{#lynus.ag#()}
	lr_EnergyCounter_EM4	: LREAL;						//{#lynus.ag#()}
	lr_EnergyCounter_EM5	: LREAL;						//{#lynus.ag#()}
	lr_EnergyCounter_EM6	: LREAL;						//{#lynus.ag#()}
	lr_EnergyCounter_House	: LREAL;						//{#lynus.ag#()}
END_VAR

// grid measurement
fbEL3443DPM(
	bEnable 	:= TRUE, 
	bInvers_CH1 := , 
	bInvers_CH2	:= , 
	bInvers_CH3	:= , 
	uiCurrentTransformerRatio:= uiCurrentTransformerRatio, 
	nSlaveAddr 	:= 1003,
	stEL3443_IO := ,
	pDpmData=> , 
	stDataEMPower=> , 
	stDataEMCounter=> , 
	stDataEMPowerRealTime=> , 
	stDataEMCounterRealTime=> );
fbEL3443DPM.stEL3443_IO.MDP5001_341_Input := stEL3443_IO.MDP5001_341_Input;
stEL3443_IO.MDP5001_341_Output	:= fbEL3443DPM.stEL3443_IO.MDP5001_341_Output;
 	
lr_RealPower_Grid 		:= fbEL3443DPM.stDataEMPower.lrPowerTotal; 	
lr_ApparentPower_Grid 	:= fbEL3443DPM.stDataEMPower.lrApparentPowerTotal;
lr_ReactivePower_Grid	:= fbEL3443DPM.stDataEMPower.lrReactivePowerTotal;
lr_Frequency_Grid		:= fbEL3443DPM.stDataEMPower.lrFrequency;
lr_Voltage_L1N			:= fbEL3443DPM.stDataEMPower.lrVoltageL1N;
lr_Voltage_L2N			:= fbEL3443DPM.stDataEMPower.lrVoltageL2N;
lr_Voltage_L3N			:= fbEL3443DPM.stDataEMPower.lrVoltageL3N;
lr_Voltage_L1L2			:= fbEL3443DPM.stDataEMPower.lrVoltageL1L2;
lr_Voltage_L2L3			:= fbEL3443DPM.stDataEMPower.lrVoltageL2L3;
lr_Voltage_L3L1			:= fbEL3443DPM.stDataEMPower.lrVoltageL3L1;
lr_EnergyCounter_Grid	:= fbEL3443DPM.stDataEMCounter.lrTotalCounterEnergy_Consumption;
lr_Current_L1			:= fbEL3443DPM.stDataEMPower.lrCurrentL1;
lr_Current_L2			:= fbEL3443DPM.stDataEMPower.lrCurrentL2;
lr_Current_L3			:= fbEL3443DPM.stDataEMPower.lrCurrentL3;
	 
fb_EL3446(
	bEnable:= TRUE , 
	bEnableVariantValues:= TRUE, 
	pDpmData:= fbEL3443DPM.pDpmData, 
	nSlaveAddr:= 1004, 
	bInvers_CH1:= b_Invers_FB3446_CH1, 
	bInvers_CH2:= b_Invers_FB3446_CH2, 
	bInvers_CH3:= b_Invers_FB3446_CH3, 
	bInvers_CH4:= b_Invers_FB3446_CH4, 
	bInvers_CH5:= b_Invers_FB3446_CH5, 
	bInvers_CH6:= b_Invers_FB3446_CH6, 
	uiCurrentTransformerRatio_CH1:= 32, 
	uiCurrentTransformerRatio_CH2:= 32, 
	uiCurrentTransformerRatio_CH3:= 32, 
	uiCurrentTransformerRatio_CH4:= 32, 
	uiCurrentTransformerRatio_CH5:= 32, 
	uiCurrentTransformerRatio_CH6:= 32, 
	uiVoltagePhaseSelector_CH1:= ui_PhaseSelector_CH1, 
	uiVoltagePhaseSelector_CH2:= ui_PhaseSelector_CH2, 
	uiVoltagePhaseSelector_CH3:= ui_PhaseSelector_CH3, 
	uiVoltagePhaseSelector_CH4:= ui_PhaseSelector_CH4, 
	uiVoltagePhaseSelector_CH5:= ui_PhaseSelector_CH5, 
	uiVoltagePhaseSelector_CH6:= ui_PhaseSelector_CH6, 
	bEnable3PhaseCH13:= FALSE, 
	bEnable3PhaseCH46:= FALSE, 
	stDataEMPowerRealTime:= fbEL3443DPM.stDataEMPowerRealTime, 
	stEL3446_IO := ,
	stDataEMPower_CH1=> , 
	stDataEMCounter_CH1=> , 
	stDataEMPowerRealTime_CH1=> , 
	stDataEMCounterRealTime_CH1=> , 
	stDataEMPower_CH2=> , 
	stDataEMCounter_CH2=> , 
	stDataEMPowerRealTime_CH2=> , 
	stDataEMCounterRealTime_CH2=> , 
	stDataEMPower_CH3=> , 
	stDataEMCounter_CH3=> , 
	stDataEMPowerRealTime_CH3=> , 
	stDataEMCounterRealTime_CH3=> , 
	stDataEMPower_CH4=> , 
	stDataEMCounter_CH4=> , 
	stDataEMPowerRealTime_CH4=> , 
	stDataEMCounterRealTime_CH4=> , 
	stDataEMPower_CH5=> , 
	stDataEMCounter_CH5=> , 
	stDataEMPowerRealTime_CH5=> , 
	stDataEMCounterRealTime_CH5=> , 
	stDataEMPower_CH6=> , 
	stDataEMCounter_CH6=> , 
	stDataEMPowerRealTime_CH6=> , 
	stDataEMCounterRealTime_CH6=> );
fb_EL3446.stEL3446_IO.MDP5001_342_Input := stEL3446_IO.MDP5001_342_Input;
stEL3446_IO.MDP5001_342_Output := 	fb_EL3446.stEL3446_IO.MDP5001_342_Output;

lrPower_EM1				:= 	LIMIT(0,fb_EL3446.stDataEMPower_CH1.lrPowerTotal,100);
lrPower_EM2				:= 	LIMIT(0,fb_EL3446.stDataEMPower_CH2.lrPowerTotal,100);
lrPower_EM3				:= 	LIMIT(0,fb_EL3446.stDataEMPower_CH3.lrPowerTotal,100);
lrPower_EM4				:= 	LIMIT(0,fb_EL3446.stDataEMPower_CH4.lrPowerTotal,100);
lrPower_EM5				:= 	LIMIT(0,fb_EL3446.stDataEMPower_CH5.lrPowerTotal,100);
lrPower_EM6				:= 	LIMIT(0,fb_EL3446.stDataEMPower_CH6.lrPowerTotal,100);
lr_EnergyCounter_EM1	:= 	fb_EL3446.stDataEMCounter_CH1.lrTotalCounterEnergy_Consumption;
lr_EnergyCounter_EM2	:= 	fb_EL3446.stDataEMCounter_CH2.lrTotalCounterEnergy_Consumption;
lr_EnergyCounter_EM3	:= 	fb_EL3446.stDataEMCounter_CH3.lrTotalCounterEnergy_Consumption;
lr_EnergyCounter_EM4	:= 	fb_EL3446.stDataEMCounter_CH4.lrTotalCounterEnergy_Consumption;
lr_EnergyCounter_EM5	:= 	fb_EL3446.stDataEMCounter_CH5.lrTotalCounterEnergy_Consumption;
lr_EnergyCounter_EM6	:= 	fb_EL3446.stDataEMCounter_CH6.lrTotalCounterEnergy_Consumption;

IF fb_EL3446.stDataEMPower_CH1.lrPowerTotal<-0.10 THEN
	m_negativePower := TRUE;
	lrTemp_EM1 := fb_EL3446.stDataEMPower_CH1.lrPowerTotal;
END_IF 
IF fb_EL3446.stDataEMPower_CH2.lrPowerTotal<-0.10 THEN
	m_negativePower := TRUE;
	lrTemp_EM2 := fb_EL3446.stDataEMPower_CH2.lrPowerTotal;
END_IF
IF fb_EL3446.stDataEMPower_CH3.lrPowerTotal<-0.10 THEN
	m_negativePower := TRUE;
	lrTemp_EM3 := fb_EL3446.stDataEMPower_CH3.lrPowerTotal;
END_IF
IF fb_EL3446.stDataEMPower_CH4.lrPowerTotal<-0.10 THEN
	m_negativePower := TRUE;
	lrTemp_EM4 := fb_EL3446.stDataEMPower_CH4.lrPowerTotal;
END_IF
IF  fb_EL3446.stDataEMPower_CH5.lrPowerTotal<-0.10 THEN
	m_negativePower := TRUE;
	lrTemp_EM5 := fb_EL3446.stDataEMPower_CH5.lrPowerTotal;
END_IF

// calculate not measured house power
lrPower_House := lr_RealPower_Grid - lrPower_EM1 - lrPower_EM2 - lrPower_EM3 - lrPower_EM4 - lrPower_EM5 - lrPower_EM6;
lrPower_House := LIMIT(0,lrPower_House,100);
fbCounter_House(	byActiveTariff:= 1, 
					lrPowerInput:= lrPower_House, 
					lrTotalCounterEnergy_Consumption=> , 
					lrTotalCounterEnergy_Production=> , 
					lrCounterEnergyT1_Consumption=> , 
					lrCounterEnergyT2_Consumption=> , 
					lrCounterEnergyT1_Production=> , 
					lrCounterEnergyT2_Production=> );
lr_EnergyCounter_House := 	fbCounter_House.lrCounterEnergyT1_Consumption;				


// transfer raw data to cloud
lrPowerTotal_raw_W_EM1				:= 		prgEM.fb_EL3446.stDataEMPowerRealTime_CH1.lrPowerTotal;
lrApparentPowerTotal_raw_VA_EM1 	:= 		prgEM.fb_EL3446.stDataEMPowerRealTime_CH1.lrApparentPowerTotal;
lrReactivePowerTotal_raw_VAr_EM1	:= 		prgEM.fb_EL3446.stDataEMPowerRealTime_CH1.lrReactivePowerTotal;
lrPowerTotal_raw_W_EM2				:= 		prgEM.fb_EL3446.stDataEMPowerRealTime_CH2.lrPowerTotal;
lrApparentPowerTotal_raw_VA_EM2 	:= 		prgEM.fb_EL3446.stDataEMPowerRealTime_CH2.lrApparentPowerTotal;
lrReactivePowerTotal_raw_VAr_EM2	:= 		prgEM.fb_EL3446.stDataEMPowerRealTime_CH2.lrReactivePowerTotal;
lrPowerTotal_raw_W_EM3				:= 		prgEM.fb_EL3446.stDataEMPowerRealTime_CH3.lrPowerTotal;
lrApparentPowerTotal_raw_VA_EM3 	:= 		prgEM.fb_EL3446.stDataEMPowerRealTime_CH3.lrApparentPowerTotal;
lrReactivePowerTotal_raw_VAr_EM3	:= 		prgEM.fb_EL3446.stDataEMPowerRealTime_CH3.lrReactivePowerTotal;
lrPowerTotal_raw_W_EM4				:= 		prgEM.fb_EL3446.stDataEMPowerRealTime_CH4.lrPowerTotal;
lrApparentPowerTotal_raw_VA_EM4 	:= 		prgEM.fb_EL3446.stDataEMPowerRealTime_CH4.lrApparentPowerTotal;
lrReactivePowerTotal_raw_VAr_EM4	:= 		prgEM.fb_EL3446.stDataEMPowerRealTime_CH4.lrReactivePowerTotal;
lrPowerTotal_raw_W_EM5				:= 		prgEM.fb_EL3446.stDataEMPowerRealTime_CH5.lrPowerTotal;
lrApparentPowerTotal_raw_VA_EM5 	:= 		prgEM.fb_EL3446.stDataEMPowerRealTime_CH5.lrApparentPowerTotal;
lrReactivePowerTotal_raw_VAr_EM5	:= 		prgEM.fb_EL3446.stDataEMPowerRealTime_CH5.lrReactivePowerTotal;

END_PROGRAM

// ---- POUs/prgSystemTime.TcPOU
PROGRAM prgSystemTime
VAR
	fbNTGetSystemTime: NT_GetTime;
	intStateSystemTime: INT;
	structSystemTime: timestruct;
	stringSystemTime: STRING(19);
	stringSystemTime_ms: STRING(23);
	stringSystemDate: STRING(10);
	stringTimeOnly_ms: STRING(12);
	stringTimeOnly: STRING(8);
	stringMonth: STRING(4);
	strTimeStampEventrecorder: STRING;
END_VAR

(* get system time *)
CASE intStateSystemTime OF
	0:	fbNTGetSystemTime(Start:=FALSE);
		intStateSystemTime:=20;
	20:	fbNTGetSystemTime(Start:=TRUE);
		intStateSystemTime:=30;
	30:	fbNTGetSystemTime();
		IF NOT fbNTGetSystemTime.BUSY THEN
			structSystemTime:=fbNTGetSystemTime.TIMESTR;
			intStateSystemTime:=40;
		END_IF
	40:	intStateSystemTime:=0;
		stringSystemTime := SYSTEMTIME_TO_STRING(IN := structSystemTime);
		stringSystemTime_ms := SYSTEMTIME_TO_STRING(IN := structSystemTime);
		stringSystemDate := SYSTEMTIME_TO_STRING(IN := structSystemTime);
		stringTimeOnly_ms:=RIGHT(stringSystemTime_ms,12);
		stringTimeOnly:=RIGHT(stringSystemTime,8);
		CASE structSystemTime.wMonth OF
			1:	stringMonth:='Jan';
			2:	stringMonth:='Feb';
			3:	stringMonth:='Mae';
			4:	stringMonth:='Apr';
			5:	stringMonth:='Mai';
			6:	stringMonth:='Jun';
			7:	stringMonth:='Jul';
			8:	stringMonth:='Aug';
			9:	stringMonth:='Sep';
			10:	stringMonth:='Okt';
			11:	stringMonth:='Nov';
			12:	stringMonth:='Dez';
		END_CASE
		strTimeStampEventrecorder := CONCAT(WORD_TO_STRING(structSystemTime.wYear),stringMonth);
		IF structSystemTime.wDay <10 THEN
			strTimeStampEventrecorder := CONCAT(strTimeStampEventrecorder,'0');
		END_IF
		strTimeStampEventrecorder := CONCAT(strTimeStampEventrecorder,WORD_TO_STRING(structSystemTime.wDay));
		strTimeStampEventrecorder := CONCAT(strTimeStampEventrecorder,' ');
		IF structSystemTime.wHour <10 THEN
			strTimeStampEventrecorder := CONCAT(strTimeStampEventrecorder,'0');
		END_IF
		strTimeStampEventrecorder := CONCAT(strTimeStampEventrecorder,WORD_TO_STRING(structSystemTime.wHour));
		strTimeStampEventrecorder := CONCAT(strTimeStampEventrecorder,':');
		IF structSystemTime.wMinute <10 THEN
			strTimeStampEventrecorder := CONCAT(strTimeStampEventrecorder,'0');
		END_IF
		strTimeStampEventrecorder := CONCAT(strTimeStampEventrecorder,WORD_TO_STRING(structSystemTime.wMinute));
		strTimeStampEventrecorder := CONCAT(strTimeStampEventrecorder,':');
		IF structSystemTime.wSecond <10 THEN
			strTimeStampEventrecorder := CONCAT(strTimeStampEventrecorder,'0');
		END_IF
		strTimeStampEventrecorder := CONCAT(strTimeStampEventrecorder,WORD_TO_STRING(structSystemTime.wSecond));
		strTimeStampEventrecorder := CONCAT(strTimeStampEventrecorder,'.');
		IF structSystemTime.wMilliseconds <10 THEN
			strTimeStampEventrecorder := CONCAT(strTimeStampEventrecorder,'00');
		ELSIF structSystemTime.wMilliseconds <100 THEN
			strTimeStampEventrecorder := CONCAT(strTimeStampEventrecorder,'0');
		END_IF
		strTimeStampEventrecorder := CONCAT(strTimeStampEventrecorder,WORD_TO_STRING(structSystemTime.wMilliseconds));
END_CASE

END_PROGRAM
